FUNCTION_BLOCK StateRequest_View
  (* Version 0.1, 2005-12-14, Oscar Ljungkrantz, Chalmers *)
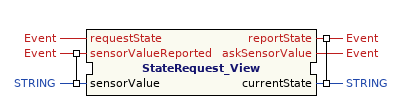
  EVENT_INPUT
    requestState;
    sensorValueReported WITH sensorValue;
  END_EVENT
  EVENT_OUTPUT
    reportState WITH currentState;
    askSensorValue;
  END_EVENT
  VAR_INPUT
    sensorValue : STRING;
  END_VAR
  VAR_OUTPUT
    currentState : STRING;
  END_VAR
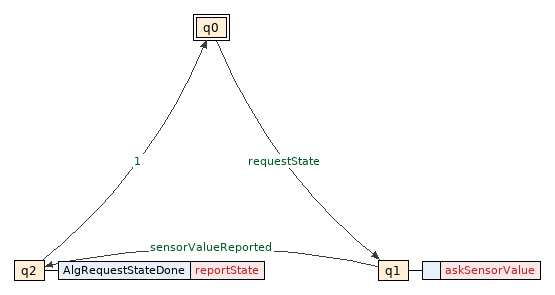
  EC_STATES
    q0;
    q1 : -> askSensorValue;
    q2 : AlgRequestStateDone -> reportState;
  END_STATES
  EC_TRANSITIONS
    q0 TO q1 := requestState;
    q1 TO q2 := sensorValueReported;
    q2 TO q0 := 1;
  END_TRANSITIONS
  ALGORITHM AlgRequestStateDone IN Java:
currentState = sensorValue;
  END_ALGORITHM
END_FUNCTION_BLOCK
(* other elements stored in the file *)
(* InternalVars> <VarDeclaration Name="" Type="" InitialValue="" /> </InternalVars *)
